// Mitsubishi GX Works2 project: z01   PLC: Q02/Q02H

PROGRAM MAIN
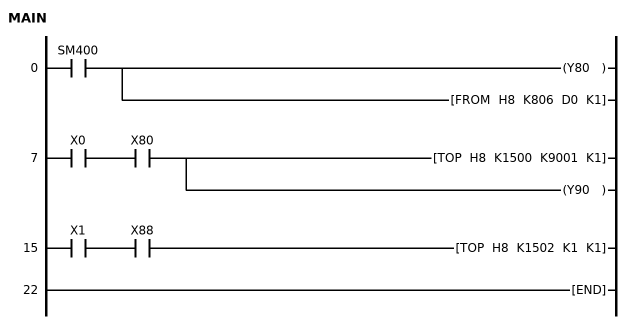
0     LD      SM400
      OUT     Y80
      FROM    H8 K806 D0 K1
7     LD      X0
      AND     X80
      TOP     H8 K1500 K9001 K1
      OUT     Y90
15    LD      X1
      AND     X88
      TOP     H8 K1502 K1 K1
22    END
END_PROGRAM
